Fanuc KAREL source: ka00155.KL

-- PROVISIONAL review KL for V770-1; original PC SHA256 1a6c9c42c5f9019b9606cb48cbcf691dee296d929fab2f1826e4db101d5bd679
-- Incomplete behavior may be omitted. Consult companion uncertainty JSON. Do not deploy.
PROGRAM KA00155
%NOLOCKGROUP
-- UNRESOLVED_DECL SRC type=002011
-- UNRESOLVED_DECL DST type=002011
BEGIN
  -- UNRESOLVED_PC offsets 5-19; opcodes 22,22,1E
  -- UNRESOLVED_PC offsets 24-28; opcodes 7F
END KA00155
